TYPE "Positioning_DOL_Machine_Manager"
VERSION : 0.1
// Block: Positioning_DOL_Machine_Manager
   STRUCT
      EnableStopDoorOpeningReq : Bool;
      EnableStopInPhase : Bool;
      EnableStopProgrammed : Bool;
      Control_ON : Bool;
      Minus : Bool;
      Plus : Bool;
      MoveToPos : Bool;
      Pos : LReal;
      Speed : LReal;
   END_STRUCT;

END_TYPE
